PROGRAM MAIN
VAR
	fbChatWindow : FB_Mediator;
	fbUsers	     : ARRAY[1..Param.MAX_COLLEAGUES] OF FB_Colleague;
	
	ChatWindow	 : I_Mediator;
	Users		 : ARRAY[1..Param.MAX_COLLEAGUES] OF I_Colleague;
	
	// Task and Demo Control
	bStartDemo	: BOOL := TRUE;
	bInit 		: BOOL := FALSE;
	i: INT;
END_VAR

IF NOT bInit THEN
	bInit := TRUE;
	// Initialize Interface to Mediator
	ChatWindow := fbChatWindow;
	FOR i := 1 TO Param.MAX_COLLEAGUES DO
		// Initialize Interface to Colleagues
		Users[i] := fbUsers[i];
		// Assign Mediator to Colleagues
		fbUsers[i](iMediator := ChatWindow);
	END_FOR
END_IF

// Assign Users 
fbChatWindow(iColleague := Users);


IF bStartDemo THEN
	bStartDemo := FALSE;
	Users[1].operation('Hi! How is everyone?');
	Users[2].operation('Good good..');
	Users[4].operation('Doing fine');
	Users[5].operation('Yup! All is well');
	Users[3].operation('I need a beer right about now');
	Users[6].operation('Had a long day?');	
	Users[3].operation('Yuuup, very long...');
END_IF

END_PROGRAM

(* stored: Version 1.1.0.1, ProductVersion 3.1.4024.12
   POU MAIN: Id {d2846f60-a5b9-420e-9422-ce267f63bc31}, SpecialFunc None *)
